Staubli VAL3: enableQueue.pgx

public program enableQueue()
// this program enables the queing of the detected objects
begin
  // this program enables the queing of the detected objects
  //
  // Created  05-01-07                            C.CURRIVAND
  //----------------------------------------------------------------
  //
  bEnableQueuing=true
  if cfg:bLog
    logMsg(sConvNum+"(enableQueue)>>Queuing of detected object enabled")
  endIf
end
